FUNCTION_BLOCK FB_Blinking
VAR_INPUT
	pVariable		:POINTER TO BOOL;		//Address of variable to blink
	interval		:TIME;					//Blink interval
END_VAR
VAR_OUTPUT
END_VAR
VAR
	bState			:BOOL;
	tonTimer		:TON;
END_VAR

tonTimer(IN:=TRUE , PT:= interval);

IF tonTimer.Q THEN 
	bState := NOT bState;
	tonTimer(IN:=FALSE, PT:= interval);
END_IF

pVariable^ := bState;

END_FUNCTION_BLOCK

(* stored: Version 1.1.0.1, ProductVersion 3.1.4022.16
   POU FB_Blinking: Id {877787ab-67ea-4a46-89ca-8d203a4a157c}, SpecialFunc None *)
